RoboDK station: UR3E_Station_Conveyor_Classify_Bolts.rdk

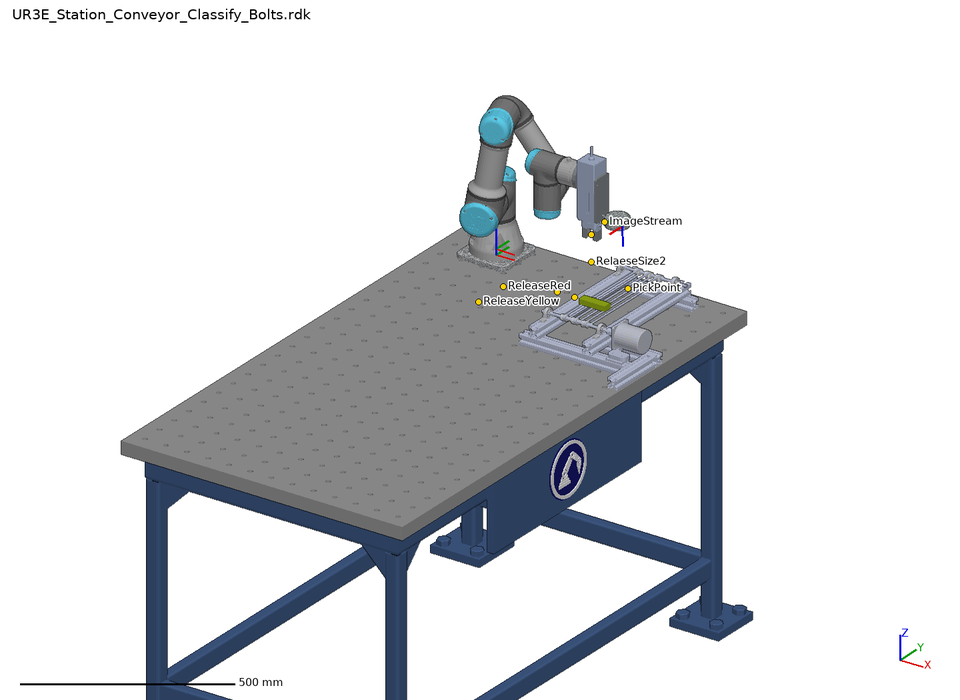
[picture v0: the station drawn from its stored meshes, robots at their saved joint values, targets as dots, program paths as lines]
Station UR3E_Station_Conveyor_Classify_Bolts (saved by RoboDK 5.2.5). Poses are relative to the parent item; angles as X-Y-Z fixed-axis rotations.
Station parameters (name, value as stored): IO_5, 1, IO_10, 0, RECORD_READY, 0, True, 0, IO_11, 0, IO_0, 0, 10, 1
  - frame World Frame at (0, 0, 0) mm
    - frame UR3e Base at (0, 0, 15) mm
      - robot UR3e: 6 axes, payload 3 kg, reach 500 mm, repeatability 0.03 mm, weight 11 kg
          modified DH rows (alpha deg, a mm, theta deg, d mm): 0, 0, 0, 151.9; 90, 0, 180, 0; 0, 243.55, 0, 0; 0, 213.2, 0, 131.05; -90, 0, 0, 85.35; 90, 0, 180, 92.1
          joint limits [-360, -360, -360, -360, -360, -360] to [360, 360, 360, 360, 360, 360]; home [0, -90, -90, 0, 90, 0]; saved at [19.746, -99.416, -136.945, 56.371, 70.253, 0]
        - tool Gripper, TCP at (0, 145, 35) mm, size 63 x 236.5 x 138.7 mm, geometry from RGI14_cBrida_UR3e.STEP
        - frame Camera Frame at (-1.25, 99.12, 122.31) mm, rotated rx -89.49 ry 0.51 rz -0.14 deg
          - camera My Camera
      - target PickPoint (Cartesian target) at (490.61, -164.44, 100.88) mm, rotated rx -90.01 ry 0 rz -90.01 deg; joints [-5.161, -149.095, -68.963, 38.044, 95.156, -0.002] of UR3e
    - object Table 1400x800x800mm at (250, -250, 0) mm, rotated rx 0 ry 0 rz -90 deg, size 1420 x 820 x 800 mm, geometry from Table-1400x800x800mm.sld
    - object Mounting_Plate_UR3e at (0, 0, 0) mm, size 140 x 140 x 15 mm, geometry from Mounting_Plate_UR3e.stp
    - target ImageStream (Cartesian target) at (400.3, -131.05, 250) mm, rotated rx -90 ry 0 rz -90 deg; joints [0, -108.893, -95.39, 24.283, 90, 0] of UR3e
    - target ReleaseRed (Cartesian target) at (234, -305, 105) mm, rotated rx -90.2 ry -0.28 rz 177.77 deg; joints [-10.677, -131.219, -108.96, 58.788, 8.448, 1.092] of UR3e
    - target ReleaseYellow (Cartesian target) at (234, -405, 105) mm, rotated rx -90.2 ry -0.28 rz 177.77 deg; joints [-28.398, -142.152, -83.03, 44.718, 26.167, 0.131] of UR3e
    - target ReleaseSize (Cartesian target) at (320, -70, 170) mm, rotated rx -90 ry 0 rz -90 deg; joints [19.746, -99.414, -136.957, 56.37, 70.251, 0] of UR3e
    - target ReleaseBolt (Cartesian target) at (250, -180, 60) mm, rotated rx -90 ry 0 rz -90 deg; joints [-18.712, -137.061, -134.054, 91.114, 108.709, 0] of UR3e
    - target ReleaseBolt2 (Cartesian target) at (300, -180, 60) mm, rotated rx -90 ry 0 rz -90 deg; joints [-14.478, -137.816, -123.567, 81.383, 104.475, 0] of UR3e
    - target ReleaseBolt1 (Cartesian target) at (350, -180, 60) mm, rotated rx -90 ry 0 rz -90 deg; joints [-11.7, -140.431, -111.245, 71.676, 101.697, 0] of UR3e
    - target RelaeseSize2 (Cartesian target) at (320, -70, 100) mm, rotated rx -90 ry 0 rz -90 deg; joints [19.746, -122.93, -140.197, 83.126, 70.251, 0] of UR3e
  - program Image_Stream_Position (3 instructions, listed below)
  - program Pick_Position (3 instructions, listed below)
  - program Gripper Open (2 instructions, listed below)
  - program Gripper Close (2 instructions, listed below)
  - program Gripper_TurnH (2 instructions, listed below)
  - program Gripper_TurnV (2 instructions, listed below)
  - program Convey_ON (1 instructions, listed below)
  - program Convey_OFF (1 instructions, listed below)
  - object Conveyor_Assembly_RoboDK at (210, 250, -220) mm, rotated rx 90 ry 0 rz 0 deg, size 330 x 105 x 467.7 mm, geometry from Conveyor_Assembly_RoboDK.STEP

--- program Image_Stream_Position (robot UR3e) ---
  Set Ref.: World Frame
  Set Tool: Gripper
  MoveJ (Target 9) -> target RelaeseSize2

--- program Pick_Position (robot UR3e) ---
  Set Ref.: World Frame
  Set Tool: Gripper
  MoveJ (PickPoint)

--- program Gripper Open (robot UR3e) ---
  Set IO_10=1
  Pause 500 ms

--- program Gripper Close (robot UR3e) ---
  Set IO_10=0
  Pause 500 ms

--- program Gripper_TurnH (robot UR3e) ---
  Set IO_11=1
  Pause 500 ms

--- program Gripper_TurnV (robot UR3e) ---
  Set IO_11=0
  Pause 500 ms

--- program Convey_ON (robot UR3e) ---
  Set IO_0=1

--- program Convey_OFF (robot UR3e) ---
  Set IO_0=0
